(* IEC 61131-3 sources: RL_MAR/experiments/comparison/autoplc/results/gpt-4o_20260511_211137/med_88, 1 file *)

(* ---- med_88_1.st ---- *)
FUNCTION_BLOCK SmartLockerControl
VAR_INPUT
    AccessCode : INT; (* Input for user access code *)
    LockerNumber : INT; (* Input for selected locker number *)
END_VAR
VAR_OUTPUT
    LockerOpen : BOOL; (* Output to control locker door *)
END_VAR
VAR
    LockerStatus : ARRAY[1..10] OF BOOL; (* Status of individual lockers: TRUE=locked, FALSE=empty *)
    LockerAccessCode : ARRAY[1..10] OF INT; (* Locker access codes *)
    i : INT; (* Loop counter *)
END_VAR

(* Initialization of LockerStatus and LockerAccessCode arrays *)
(* This initialization should be done once, typically in a constructor or initialization routine *)
FOR i := 1 TO 10 DO
    LockerStatus[i] := TRUE; (* Initially, all lockers are locked *)
END_FOR

LockerAccessCode[1] := 1234;
LockerAccessCode[2] := 5678;
LockerAccessCode[3] := 9876;
LockerAccessCode[4] := 4321;
LockerAccessCode[5] := 6543;
LockerAccessCode[6] := 7890;
LockerAccessCode[7] := 3456;
LockerAccessCode[8] := 8765;
LockerAccessCode[9] := 2345;
LockerAccessCode[10] := 6789;

(* Access Control Logic *)
IF (LockerNumber >= 1) AND (LockerNumber <= 10) THEN
    IF (AccessCode = LockerAccessCode[LockerNumber]) THEN
        LockerOpen := TRUE; (* Open the locker *)
        LockerStatus[LockerNumber] := FALSE; (* Update status to unlocked *)
    ELSE
        LockerOpen := FALSE; (* Do not open the locker if access code is incorrect *)
    END_IF
ELSE
    LockerOpen := FALSE; (* Invalid locker number, do not open any locker *)
END_IF

END_FUNCTION_BLOCK
